FUNCTION_BLOCK List_TEST
VAR
	List  : List<5>;
	Item1 : Item_Mockup;
	Item2 : Item_Mockup;
	Item3 : Item_Mockup;
END_VAR

InsertByIndex();
InsertByIndexFail();
InsertByIndexShift();
GetByIndex();
ContainsItemTrue();
ContainsItemFalse();
RemoveItemByIndex();
Clear();
AddTwoItems();
RemoveFirstItem();
RemoveLastItem();
RemoveToEmpty();
ContainsAfterItemRemoval();
RemoveDuplicateItems();
ContainsOnEmptyList();
Test();
InsertIndex0Shift();

METHOD AddTwoItems
VAR_INST
	Expected : UDINT;
	Actual	 : UDINT;
END_VAR
IF TestSuite.Test(__POUNAME()).ExecuteTest() THEN
	Expected := 2;
	List.Clear();
	List.AddItem(Item1);
	List.AddItem(Item2);
	Actual := List.Count;
	List.AddItem(Item3);
	TestSuite.Test(__POUNAME()).AssertEqual(Expected, Actual);
END_IF
END_METHOD

METHOD Clear
VAR
	Expected : UDINT;
	Actual	 : UDINT;
END_VAR
IF TestSuite.Test(__POUNAME()).ExecuteTest() THEN
	Expected := 0;
	List.Clear();
	Actual := List.Count;
	TestSuite.Test(__POUNAME()).AssertEqual(Expected, Actual);
END_IF
END_METHOD

METHOD ContainsAfterItemRemoval
VAR
	Expected	 : BOOL;
	Actual		 : BOOL;
	ExpectedItem : I_Base;
	ActualItem	 : I_Base;
END_VAR
IF TestSuite.Test(__POUNAME()).ExecuteTest() THEN
	Expected	 := TRUE;
	ExpectedItem := Item2;
	List.Clear();
	ExpectedItem := Item2;
	List.AddItem(Item1);
	List.AddItem(Item2);
	List.RemoveItem(Item1);
	ActualItem := List.GetAtIndex(0);
	Actual	   := ExpectedItem = ActualItem;
	TestSuite.Test(__POUNAME()).AssertEqual(Expected, Actual);

	//cleanup
	List.Clear();
END_IF
END_METHOD

METHOD ContainsItemFalse
VAR
	Expected : BOOL;
	Actual	 : BOOL;
END_VAR
IF TestSuite.Test(__POUNAME()).ExecuteTest() THEN
	Expected := FALSE;
	Actual	 := List.ContainsItem(Item3);
	TestSuite.Test(__POUNAME()).AssertEqual(Expected, Actual);
END_IF
END_METHOD

METHOD ContainsItemTrue
VAR
	Expected : BOOL;
	Actual	 : BOOL;
END_VAR
IF TestSuite.Test(__POUNAME()).ExecuteTest() THEN
	Expected := TRUE;
	Actual	 := List.ContainsItem(Item2);
	TestSuite.Test(__POUNAME()).AssertEqual(Expected, Actual);
END_IF
END_METHOD

METHOD ContainsOnEmptyList
VAR
	Expected : BOOL;
	Actual	 : BOOL;
END_VAR
IF TestSuite.Test(__POUNAME()).ExecuteTest() THEN
	Expected := FALSE;
	List.Clear();
	Actual := List.ContainsItem(Item1);
	TestSuite.Test(__POUNAME()).AssertEqual(Expected, Actual);
END_IF
END_METHOD

METHOD GetByIndex
VAR
	Expected   : BOOL;
	Actual	   : BOOL;
	TargetItem : I_Base;
	ActualItem : I_Base;
END_VAR
IF TestSuite.Test(__POUNAME()).ExecuteTest() THEN
	Expected   := TRUE;
	TargetItem := Item2;
	ActualItem := List.GetAtIndex(1);
	Actual	   := TargetItem = ActualItem;
	TestSuite.Test(__POUNAME()).AssertEqual(Expected, Actual);
END_IF
END_METHOD

METHOD InsertByIndex
VAR
	Expected   : UDINT;
	Actual	   : UDINT;
	TargetItem : I_Base;
	ActualItem : I_Base;
END_VAR
IF TestSuite.Test(__POUNAME()).ExecuteTest() THEN
	Expected := 1;
	List.InsertAtIndex(Item2, 0);
	Actual := List.Count;
	TestSuite.Test(__POUNAME()).AssertEqual(Expected, Actual);
END_IF
END_METHOD

METHOD InsertByIndexFail
VAR
	Expected : BOOL;
	Actual	 : BOOL;
END_VAR
IF TestSuite.Test(__POUNAME()).ExecuteTest() THEN
	Expected := FALSE;
	Actual	 := List.InsertAtIndex(Item2, 2);
	TestSuite.Test(__POUNAME()).AssertEqual(Expected, Actual);
END_IF
END_METHOD

METHOD InsertByIndexShift
VAR
	Expected   : UDINT;
	Actual	   : UDINT;
	TargetItem : I_Base;
	ActualItem : I_Base;
END_VAR
IF TestSuite.Test(__POUNAME()).ExecuteTest() THEN
	Expected := 2;
	List.InsertAtIndex(Item1, 0);
	Actual := List.Count;
	TestSuite.Test(__POUNAME()).AssertEqual(Expected, Actual);
END_IF
END_METHOD

METHOD InsertIndex0Shift
VAR
	Expected	  : BOOL;
	Actual		  : BOOL;
	ExpectedItems : ARRAY[0..4] OF I_Base;
	ActualItems	  : ARRAY[0..4] OF I_Base;
	Item4		  : Item_Mockup;
	Item5		  : Item_Mockup;
	i			  : UDINT;
END_VAR
IF TestSuite.Test(__POUNAME()).ExecuteTest() THEN
	Expected		 := TRUE;
	ExpectedItems[0] := Item5;
	ExpectedItems[1] := Item1;
	ExpectedItems[2] := Item2;
	ExpectedItems[3] := Item3;
	ExpectedItems[4] := Item4;
	List.Clear();
	FOR i := 1 TO 4 DO
		List.AddItem(ExpectedItems[i]);
	END_FOR

	List.InsertAtIndex(Item5, 0);
	Actual := TRUE;
	FOR i := 0 TO 4 DO
		ActualItems[i] := List.GetAtIndex(i);
		Actual		   := Actual AND ExpectedItems[i] = ActualItems[i];
	END_FOR

	TestSuite.Test(__POUNAME()).AssertEqual(Expected, Actual);

	//cleanup
	List.Clear();
END_IF
END_METHOD

METHOD RemoveDuplicateItems
VAR
	Expected   : UDINT;
	Actual	   : UDINT;
	TargetItem : I_Base;
	ActualItem : I_Base;
END_VAR
IF TestSuite.Test(__POUNAME()).ExecuteTest() THEN
	Expected   := 1;
	TargetItem := Item2;
	List.Clear();
	List.AddItem(Item1);
	List.AddItem(Item1);
	List.AddItem(Item2);
	List.RemoveItem(Item1);
	Actual := List.Count;
	TestSuite.Test(__POUNAME()).AssertEqual(Expected, Actual);

	//cleanup
	List.Clear();
END_IF
END_METHOD

METHOD RemoveFirstItem
VAR_INST
	Expected   : BOOL;
	Actual	   : BOOL;
	TargetItem : I_Base;
	ActualItem : I_Base;
END_VAR
IF TestSuite.Test(__POUNAME()).ExecuteTest() THEN
	Expected   := TRUE;
	TargetItem := Item2;
	List.RemoveItem(Item1);
	ActualItem := List.GetAtIndex(0);
	Actual	   := (TargetItem = ActualItem) AND (List.Count = 2);
	TestSuite.Test(__POUNAME()).AssertEqual(Expected, Actual);
END_IF
END_METHOD

METHOD RemoveItemByIndex
VAR
	Expected   : UDINT;
	Actual	   : UDINT;
	TargetItem : I_Base;
	ActualItem : I_Base;
END_VAR
IF TestSuite.Test(__POUNAME()).ExecuteTest() THEN
	Expected := 1;
	List.RemoveAtIndex(1);
	Actual := List.Count;
	TestSuite.Test(__POUNAME()).AssertEqual(Expected, Actual);
END_IF
END_METHOD

METHOD RemoveLastItem
VAR_INST
	Expected   : BOOL;
	Actual	   : BOOL;
	TargetItem : I_Base;
	ActualItem : I_Base;
END_VAR
IF TestSuite.Test(__POUNAME()).ExecuteTest() THEN
	Expected   := TRUE;
	TargetItem := 0;
	List.RemoveItem(Item3);
	ActualItem := List.GetAtIndex(2);
	Actual	   := (TargetItem = ActualItem) AND (List.Count = 1);
	TestSuite.Test(__POUNAME()).AssertEqual(Expected, Actual);
END_IF
END_METHOD

METHOD RemoveToEmpty
VAR_INST
	Expected : UDINT;
	Actual	 : UDINT;
END_VAR
IF TestSuite.Test(__POUNAME()).ExecuteTest() THEN
	Expected := 0;
	List.RemoveItem(Item2);
	Actual := List.Count;
	TestSuite.Test(__POUNAME()).AssertEqual(Expected, Actual);
END_IF
END_METHOD

METHOD Test
VAR
	Expected	 : BOOL;
	Actual		 : BOOL;
	ExpectedItem : I_Base;
	ActualItem	 : I_Base;
END_VAR
IF TestSuite.Test(__POUNAME()).ExecuteTest() THEN
	Expected	 := TRUE;
	ExpectedItem := Item2;
	List.Clear();
	List.AddItem(Item1);
	List.AddItem(Item2);
	List.RemoveAtIndex(0);
	ActualItem := List.GetAtIndex(0);
	Actual	   := ActualItem = ExpectedItem;
	TestSuite.Test(__POUNAME()).AssertEqual(Expected, Actual);

	//cleanup
	List.Clear();
END_IF
END_METHOD

END_FUNCTION_BLOCK

(* stored: Version 1.1.0.1, ProductVersion 3.1.4026.18
   POU List_TEST: Id {a848f4ac-0118-45a2-9c47-c6777ed9c090}, SpecialFunc None
   Method AddTwoItems: Id {6b8278f7-507e-4816-8aa2-6e0605d211be}
   Method Clear: Id {afebee15-fb3d-4322-a9d8-5ea7b0c92591}
   Method ContainsAfterItemRemoval: Id {1a680b26-74e2-4ded-82c9-dd0d331ec684}
   Method ContainsItemFalse: Id {f9bbecf9-ba00-4638-80f2-4044955d76fe}
   Method ContainsItemTrue: Id {76c58a44-02b6-43d6-a77c-d722386ec806}
   Method ContainsOnEmptyList: Id {eefb6ace-2f99-4090-90a0-410ba8def1b9}
   Method GetByIndex: Id {698dd518-d288-414e-837b-4d9b16dd76b7}
   Method InsertByIndex: Id {7c1691d2-d493-4c25-a470-a513230c65a0}
   Method InsertByIndexFail: Id {b07346ce-10f2-4261-b88f-d36496b782fc}
   Method InsertByIndexShift: Id {d05a2f82-0fbd-4668-954f-a7a6551b722f}
   Method InsertIndex0Shift: Id {f7906ceb-2488-4ada-927d-cf7e357086ea}
   Method RemoveDuplicateItems: Id {a123a4c7-ff61-43a7-a23a-86ec6413621f}
   Method RemoveFirstItem: Id {d7314714-9304-44df-b9d3-4b51cffff581}
   Method RemoveItemByIndex: Id {ee4600d1-f3f2-4c1f-8370-8828504de452}
   Method RemoveLastItem: Id {22bd23f1-8a23-4f8d-a592-21bf3e4ff4f1}
   Method RemoveToEmpty: Id {75a8aa59-d684-4ca1-a48d-66ef396bdc81}
   Method Test: Id {0d174a6b-9247-4470-8884-0326d34f7a4a} *)
